RoboDK station: Program_VDL_Testobject_AMR_mapped.rdk

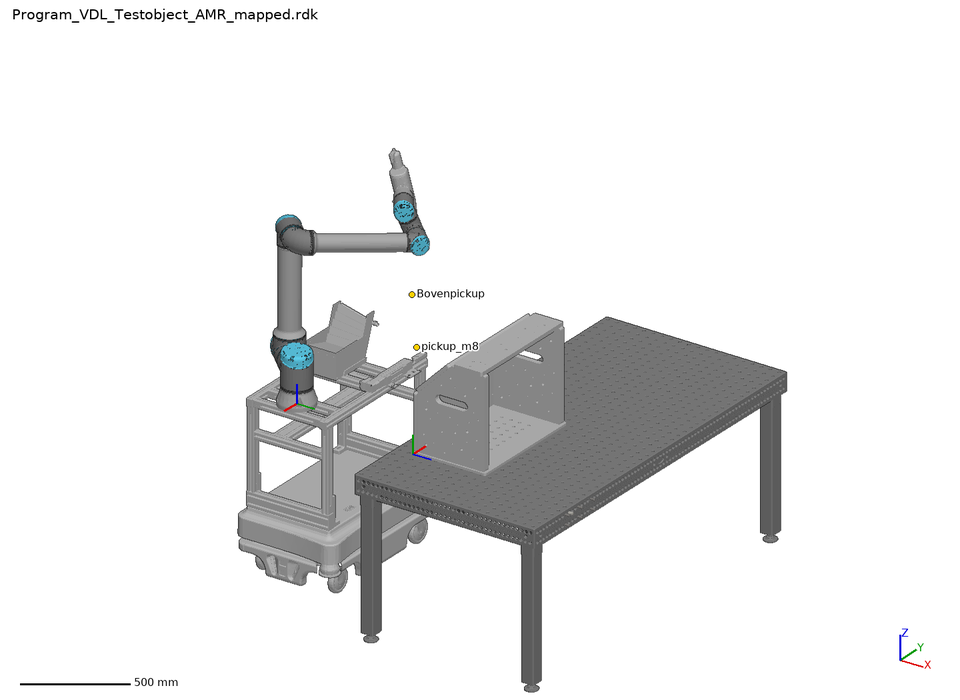
[picture v0: the station drawn from its stored meshes, robots at their saved joint values, targets as dots, program paths as lines]
Station Program_VDL_Testobject_AMR_mapped (saved by RoboDK 5.9.6). Poses are relative to the parent item; angles as X-Y-Z fixed-axis rotations.
Station parameters (name, value as stored): CollisionFreePlanner, UR10e, CollisionFreePlanner-Rob UR10e, Simplify-Mesh-Settings
  - object Lastafel at (0, 0, 0) mm, size 1021.8 x 2000 x 842 mm
  - object Lastafel_simplified at (0, 0, 0) mm, size 1000 x 2000 x 802.1 mm
  - frame UR10e Base at (-1574.73, 215.14, 116.62) mm, rotated rx 0 ry 0 rz -90 deg
    - robot UR10e: 6 axes, payload 10 kg, reach 1300 mm, repeatability 0.05 mm, weight 28.9 kg
        modified DH rows (alpha deg, a mm, theta deg, d mm): 0, 0, 0, 180.7; 90, 0, 180, 0; 0, 612.6, 0, 0; 0, 571.335, 0, 174.15; -90, 0, 0, 119.85; 90, 0, 180, 116.55
        joint limits [-180, -100, -30, -180, -180, -180] to [0, 0, 180, 180, 180, 180]; home [30.872, -95.296, 116.362, -22.187, 121.11, 179.827]; saved at [-43.827, -89.767, 94.875, 154.214, -10.442, -82.082]
      - tool schroevendraaier all in met nieuw kopstuk en tool, TCP at (210, -1, 100.6) mm, rotated rx 90 ry -90 rz 90 deg, size 86.2 x 139.7 x 345.9 mm, geometry from schroevendraaier all in met nieuw kopstuk en tool.STEP
      - tool tool simplified, TCP at (210, -1, 100.6) mm, rotated rx 90 ry -90 rz 90 deg, size 86.3 x 139.7 x 346 mm
    - object Assembly mir + frame aangepast naar ur10e versie 2 at (-733.08, 277.19, -552.66) mm, rotated rx 90 ry 0 rz 0.45 deg, size 901.1 x 1139.6 x 580.4 mm, geometry from Assembly mir + frame aangepast naar ur10e versie 2.STEP
    - object Mir + frame simplified at (-733.08, 277.19, -552.66) mm, rotated rx 90 ry 0 rz 0.45 deg, size 925.7 x 1139.7 x 582 mm
  - frame CSV Frame at (-919, 200, 49.99) mm, rotated rx 90 ry 0 rz 90.11 deg
    - object Test object at (0, 0.01, 0) mm, size 650 x 517 x 400 mm, geometry from Test object.STEP
    - object Test object simplified at (0, 0.01, 0) mm, size 650.1 x 517 x 436.5 mm
    - target pickup_m8 (joint target) at (672.95, 143.93, -450.44) mm, rotated rx 9.58 ry 86.75 rz -77.13 deg; joints [-45.747, -65.18, 99.078, -38.37, -45.221, -90.148] of UR10e
    - target Bovenpickup (joint target) at (657.59, 413.07, -465.55) mm, rotated rx 9.58 ry 86.75 rz -77.13 deg; joints [-45.787, -76.28, 85.202, -13.391, -45.26, -90.153] of UR10e
